(* Logix 5000 project; controller Project vendor 1 type 14 code 92 rev 37.11; software revision 37.00 *)

TASK MainTask (continuous, watchdog 500 ms) : MainProgram

MODULES
   Local : vendor 1 type 14 code 92 (ICP 0, rev 37.11)
END_MODULES

PROGRAM MainProgram   (* main routine MainRoutine *)
VAR
   input : BOOL;
   next_input : BOOL;
   output_1 : BOOL;
END_VAR

ROUTINE MainRoutine   (* ladder *)
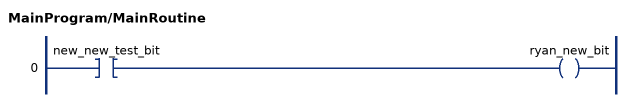
   0: XIC(new_new_test_bit)OTE(ryan_new_bit);
END_ROUTINE
END_PROGRAM
